PROGRAM LadderLogic
VAR
	ExternalILK: BOOL;
END_VAR

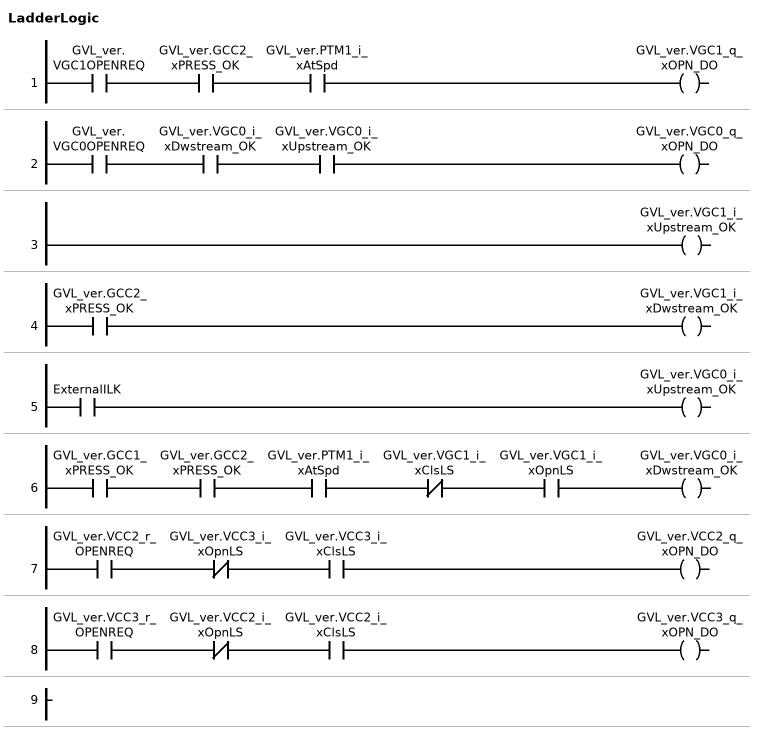
// NETWORK 1
GVL_ver.VGC1_q_xOPN_DO := GVL_ver.VGC1OPENREQ AND GVL_ver.GCC2_xPRESS_OK AND GVL_ver.PTM1_i_xAtSpd;

// NETWORK 2
GVL_ver.VGC0_q_xOPN_DO := GVL_ver.VGC0OPENREQ AND GVL_ver.VGC0_i_xDwstream_OK AND GVL_ver.VGC0_i_xUpstream_OK;

// NETWORK 3
GVL_ver.VGC1_i_xUpstream_OK := TRUE;

// NETWORK 4
GVL_ver.VGC1_i_xDwstream_OK := GVL_ver.GCC2_xPRESS_OK;

// NETWORK 5
GVL_ver.VGC0_i_xUpstream_OK := ExternalILK;

// NETWORK 6
GVL_ver.VGC0_i_xDwstream_OK := GVL_ver.GCC1_xPRESS_OK AND GVL_ver.GCC2_xPRESS_OK AND GVL_ver.PTM1_i_xAtSpd AND NOT GVL_ver.VGC1_i_xClsLS AND GVL_ver.VGC1_i_xOpnLS;

// NETWORK 7
GVL_ver.VCC2_q_xOPN_DO := GVL_ver.VCC2_r_OPENREQ AND NOT GVL_ver.VCC3_i_xOpnLS AND GVL_ver.VCC3_i_xClsLS;

// NETWORK 8
GVL_ver.VCC3_q_xOPN_DO := GVL_ver.VCC3_r_OPENREQ AND NOT GVL_ver.VCC2_i_xOpnLS AND GVL_ver.VCC2_i_xClsLS;

// NETWORK 9

END_PROGRAM

(* stored: Version 1.1.0.1, ProductVersion 3.1.4022.3
   POU LadderLogic: Id {c015a5cc-e651-4922-8201-5e6ec86c89a5}, SpecialFunc None *)
